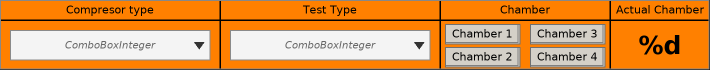
VISUALIZATION vTestPicker  // 710x70
VAR_IN_OUT
	iCompressorPick : nCompresorTypes;
	iTestType		: nTestType;
	iActualChamber	: INT;
	arControl		: ARRAY[0..3] OF stControl;
END_VAR
    Rectangle (0,20 220x50)
    ComboBoxInteger (10,30 200x30), variable: iCompressorPick, input disabled if: arControl[iActualChamber].bChamberBusy OR arControl[iActualChamber].bStartPerform, text list: 'txlCompresorTypes'
    Rectangle (0,0 220x20), "Compresor type"
    Rectangle (220,20 220x50)
    Rectangle (220,0 220x20), "Test Type"
    ComboBoxInteger (230,30 200x30), variable: iTestType, input disabled if: arControl[iActualChamber].bChamberBusy OR arControl[iActualChamber].bStartPerform, text list: 'txlTestTypes'
    Rectangle (440,0 170x20), "Chamber"
    Rectangle (440,20 170x50)
    Rectangle (610,0 100x20), "Actual Chamber"
    Rectangle (610,20 100x50), "%d", text variable: iActualChamber + 1
    Button (445,24 75x20), "Chamber 1"
        OnMouseClick: execute { iActualChamber := 0; }
    Button (530,24 75x20), "Chamber 3"
        OnMouseClick: execute { iActualChamber := 2; }
    Button (445,47 75x20), "Chamber 2"
        OnMouseClick: execute { iActualChamber := 1; }
    Button (530,47 75x20), "Chamber 4"
        OnMouseClick: execute { iActualChamber := 3; }
END_VISUALIZATION

(* stored: Version 1.1.0.1, ProductVersion 3.1.4024.12
   Visu vTestPicker: Id {ba99d946-cd4f-4b7e-a401-245b1fe80452} *)
